TYPE ST_PNInput_ACDCCharger :
STRUCT
	w_Control			:	WORD;
	ui_ACCurrentlimit	:	UINT	:=	0;
	UI_Pset				:	UINT	:=	0;
	ui_SocMaxLimit		:	UINT	:=	100;
	ui_MinGridVoltage	:	Uint	:=	360;
END_STRUCT
END_TYPE

(* stored: Version 1.1.0.1, ProductVersion 3.1.4026.18
   DUT ST_PNInput_ACDCCharger: Id {b83f44b6-9f45-4ef6-9122-b3d791f071de} *)
